// TwinCAT 3 PLC project Test
// ProgramVersion: 3.1.4024.0
// libraries:
//   Tc2_Standard, * (Beckhoff Automation GmbH)
//   Tc2_System, * (Beckhoff Automation GmbH)
//   Tc3_Module, * (Beckhoff Automation GmbH)
//   TcPiper, * (Loupe)
//   TcPluginFramework, * (Loupe)
// project tree:
//   / PlcTask.TcTTO
//   POUs/ Piper_EM.TcPOU, MAIN.TcPOU, TaskFB.TcPOU
// real-time tasks:
//   TASK PlcTask: cycle T#10ms, priority 20, ADS port 350

CONFIGURATION Test
    RESOURCE PLC ON TwinCAT3
        TASK PlcTask(INTERVAL := T#10ms, PRIORITY := 20);
        PROGRAM MAIN WITH PlcTask : MAIN;
    END_RESOURCE
END_CONFIGURATION

// ---- POUs/MAIN.TcPOU
PROGRAM MAIN
VAR
	machine_level_piper : Piper();
	task_fb : TaskFB();
	piper_em : Piper_EM(machine_level_piper, task_fb);
END_VAR

machine_level_piper();
task_fb();
piper_em();

END_PROGRAM

// ---- POUs/TaskFB.TcPOU
FUNCTION_BLOCK TaskFB EXTENDS TaskBase 
VAR_INPUT
END_VAR
VAR_OUTPUT
END_VAR
VAR
END_VAR

END_FUNCTION_BLOCK

// ---- POUs/Piper_EM.TcPOU
FUNCTION_BLOCK Piper_EM EXTENDS PiperModule
VAR_INPUT
END_VAR
VAR_OUTPUT
END_VAR
VAR
	task: REFERENCE TO TaskFB;
END_VAR

METHOD FB_init : BOOL
VAR_INPUT
	bInitRetains : BOOL; // if TRUE, the retain variables are initialized (warm start / cold start)
	bInCopyCode : BOOL;  // if TRUE, the instance afterwards gets moved into the copy code (online change)
	machineIn : REFERENCE TO Piper;
	taskFB : REFERENCE TO TaskFB;
//	context : IPluginRunner;
END_VAR
THIS^.setContext(taskFB);
task REF= taskFB;
END_METHOD

END_FUNCTION_BLOCK
